// TIA Portal V18 export
VAR_GLOBAL   // PLC tag table "04_8 Costanti Nomi Attuatore Stz08"
END_VAR
VAR_GLOBAL CONSTANT   // user constants
   M301 : Int := 1;   // Motore profila
   M365 : Int := 2;   // Motore estrattore
   EVRMRI22 : Int := 3;   // EV Salita/discesa ruota metrica per profilo RI22
   EVRMR996 : Int := 4;   // EV Salita/discesa ruota metrica per profilo R996
   EVAOS : Int := 5;   // EV lubrificazione AOS
   EVSTPR996A : Int := 6;   // EV stampo di allargatura per articolo R996
   EVSTPR996T : Int := 7;   // EV stampo di taglio per articolo R996
   EVSTPRI22T : Int := 8;   // EV stampo di taglio per articolo RI22
   EVTRASLA : Int := 9;   // EV per traslare basamento profila
END_VAR
